(* CODESYS project twinCellBalancedProduction.export

Project tree, tasks and I/O mapping:
  Device : CODESYS Control Win V3 x64, CODESYS, version 3.5.22.30
    application Application
      libraries: Standard, 3.5.22.0 (System)
      task MainTask (cyclic, interval t#20ms, priority 1) calls PLC_PRG
      data type E_MachiningCellState
      data type E_PairCoordinatorState
      global variables Commands
      global variables FIO
      function block FB_MachiningCell [ST]
      function block FB_OperatorControl [ST]
      function block FB_PairCoordinator [ST]
      function block FB_ThroughputCounter [ST]
      program PLC_PRG [ST]
      Symbols
*)

// Device/Application/E_MachiningCellState
{attribute 'qualified_only'}
{attribute 'strict'}
TYPE E_MachiningCellState :
(
    Stopped          := 0,
    Ready            := 10,
    FeedingRaw       := 20,
    WaitingForPickup := 30,
    Processing       := 40,
    Complete         := 50,
    Faulted          := 900
);
END_TYPE

// Device/Application/E_PairCoordinatorState
{attribute 'qualified_only'}
{attribute 'strict'}
TYPE E_PairCoordinatorState :
(
    Stopped          := 0,
    Ready            := 10,
    WaitPairComplete := 20,
    MergeClearance   := 30,
    Faulted          := 900
);
END_TYPE

// Device/Application/Commands
{attribute 'qualified_only'}
VAR_GLOBAL
    // Temporary operator controls from the CODESYS watch list.
    // These can later be written by an HMI without changing the plant logic.
    xStartPB : BOOL;
    xStopPB  : BOOL;
    xResetPB : BOOL;
END_VAR

// Device/Application/FIO
{attribute 'qualified_only'}
VAR_GLOBAL
    // =========================================================
    // INPUTS FROM FACTORY I/O — Factory I/O writes, PLC reads
    // =========================================================

    // Lid machining cell
    xLidsAtEntry          : BOOL;
    xLidsAtExit           : BOOL;
    xLidsCenterBusy       : BOOL;
    xLidsCenterHasError   : BOOL;
    xLidsCenterOpened     : BOOL;
    diLidsCenterProgress  : DINT;

    // Base machining cell
    xBasesAtEntry         : BOOL;
    xBasesAtExit          : BOOL;
    xBasesCenterBusy      : BOOL;
    xBasesCenterHasError  : BOOL;
    xBasesCenterOpened    : BOOL;
    diBasesCenterProgress : DINT;
	
	// Total parts processed to removal stage
	diTotalPartsCounterDisplay : DINT;
	xTotalPartsAtRemoval       : BOOL;
	
	// Twin Cell operator-panel inputs
	xTwinCellAutoModeSelected   : BOOL;
	xTwinCellEmergencyStop      : BOOL;
	xTwinCellManualModeSelected : BOOL;
	xTwinCellResetPB            : BOOL;
	xTwinCellStartPB            : BOOL;
	xTwinCellStopPB             : BOOL;

    // Factory I/O simulation status
    xFactoryIOPaused    : BOOL;
    xFactoryIOReset     : BOOL;
    xFactoryIORunning   : BOOL;
    rFactoryIOTimeScale : REAL;


    // =========================================================
    // OUTPUTS TO FACTORY I/O — PLC writes, Factory I/O reads
    // =========================================================

    // Lid machining cell
    xLidsCenterProduceLidsCmd : BOOL;
    xLidsCenterStartCmd       : BOOL;
    xLidsCenterStopCmd        : BOOL;
    xLidsCenterResetCmd       : BOOL;
    xLidsEmitterCmd           : BOOL;
    xLidsRawConveyorCmd       : BOOL;
    xLidsExitConveyor1Cmd     : BOOL;
    xLidsExitConveyor2Cmd     : BOOL;
    diLidsCounterDisplay      : DINT;

    // Base machining cell
    xBasesCenterProduceLidsCmd : BOOL;
    xBasesCenterStartCmd       : BOOL;
    xBasesCenterStopCmd        : BOOL;
    xBasesCenterResetCmd       : BOOL;
    xBasesEmitterCmd           : BOOL;
    xBasesRawConveyorCmd       : BOOL;
    xBasesExitConveyor1Cmd     : BOOL;
    xBasesExitConveyor2Cmd     : BOOL;
    diBasesCounterDisplay      : DINT;

    // Shared outfeed
    xExitConveyorCmd : BOOL;
    xRemoverCmd      : BOOL;

    // Optional Factory I/O simulation control
    diFactoryIOCameraPositionCmd : DINT;
    xFactoryIOPauseCmd           : BOOL;
    xFactoryIOResetCmd           : BOOL;
    xFactoryIORunCmd             : BOOL;
	
	// Twin Cell operator-panel outputs
	diTwinCellBasesCounterDisplay : DINT;
	diTwinCellLidsCounterDisplay  : DINT;
	
	xTwinCellResetLightCmd        : BOOL;
	xTwinCellStartLightCmd        : BOOL;
	xTwinCellStopLightCmd         : BOOL;
END_VAR

// Device/Application/PLC_PRG
PROGRAM PLC_PRG
VAR
    // Function-block instances
    fbOperator    : FB_OperatorControl;
    fbCoordinator : FB_PairCoordinator;
    fbLidsCell    : FB_MachiningCell;
    fbBasesCell   : FB_MachiningCell;
	fbStopOutfeedClearance : TON;
	fbThroughputCounter : FB_ThroughputCounter;


    // Plant-level control
    xEnablePlant              : BOOL;
	xPlantFaulted             : BOOL;
	xRecoveryResetRequired    : BOOL;
	xResetPulse               : BOOL;
	xResetRequired            : BOOL;
	xRunLatched               : BOOL;
	xStopPending              : BOOL;


    // Coordinator handshakes
    xLidsRequest  : BOOL;
    xBasesRequest : BOOL;

    xLidsReady  : BOOL;
    xBasesReady : BOOL;

    xLidsDone  : BOOL;
    xBasesDone : BOOL;


    // Fault aggregation
    xLidsFaulted       : BOOL;
    xBasesFaulted      : BOOL;
    xCoordinatorFaulted : BOOL;

    uiLidsFaultCode  : UINT;
    uiBasesFaultCode : UINT;


    // Machining-centre commands
    xLidsProduceLidsCmd  : BOOL;
    xLidsStartCmd        : BOOL;
    xLidsStopCmd         : BOOL;
    xLidsResetCmd        : BOOL;
    xLidsRawConveyorCmd  : BOOL;

    xBasesProduceLidsCmd : BOOL;
    xBasesStartCmd       : BOOL;
    xBasesStopCmd        : BOOL;
    xBasesResetCmd       : BOOL;
    xBasesRawConveyorCmd : BOOL;


    // Production totals
    diLidsCount      : DINT;
    diBasesCount     : DINT;
    diPairsCompleted : DINT;
	diTotalPartsCount : DINT;


    // Online state diagnostics
    eLidsState :
        E_MachiningCellState;

    eBasesState :
        E_MachiningCellState;

    eCoordinatorState :
        E_PairCoordinatorState;
END_VAR

// =============================================================
// 1. PLANT FAULT STATUS FROM THE PREVIOUS PLC SCAN
// =============================================================

xPlantFaulted :=
    xBasesFaulted
    OR xCoordinatorFaulted
    OR xLidsFaulted;

// Preserve the pre-reset recovery requirement for the complete
// 500 ms reset pulse.
IF NOT xResetPulse THEN
    xRecoveryResetRequired :=
        xResetRequired;
END_IF;

// =============================================================
// 2. TWIN CELL OPERATOR CONTROL
// =============================================================
// The final counter sensor is positioned immediately before
// removal. Wait until both expected parts have passed it,
// the sensor has cleared, and the outfeed has run for another
// two seconds before completing a controlled stop.

fbStopOutfeedClearance(
    IN :=
        xStopPending
        AND (eCoordinatorState = E_PairCoordinatorState.Ready)
        AND (diTotalPartsCount >= (diPairsCompleted * DINT#2))
        AND FIO.xTotalPartsAtRemoval,
    PT :=
        T#2S
);

fbOperator(
    xAutoModeSelected :=
        FIO.xTwinCellAutoModeSelected,

    xEmergencyStop :=
        NOT FIO.xTwinCellEmergencyStop,

    xFactoryIOPaused :=
        FIO.xFactoryIOPaused,

    xFactoryIORunning :=
        FIO.xFactoryIORunning,

    xManualModeSelected :=
        FIO.xTwinCellManualModeSelected,

    xPlantFaulted :=
        xPlantFaulted,

    xResetPB :=
        Commands.xResetPB
        OR FIO.xFactoryIOReset
        OR FIO.xTwinCellResetPB,

    xSafeToStop :=
    	fbStopOutfeedClearance.Q,

    xStartPB :=
        Commands.xStartPB
        OR FIO.xTwinCellStartPB,

    xStopPB :=
        Commands.xStopPB
        OR NOT FIO.xTwinCellStopPB,

    xEnablePlant =>
        xEnablePlant,

    xResetPulse =>
        xResetPulse,

    xResetRequired =>
        xResetRequired,

    xRunLatched =>
        xRunLatched,

    xStopPending =>
        xStopPending
);

// =============================================================
// 3. PAIRED-PRODUCTION COORDINATOR
// =============================================================

fbCoordinator(
    xEnable :=
        xEnablePlant,

    xReset :=
        xResetPulse,

    xAnyFault :=
        xLidsFaulted
        OR xBasesFaulted,

    xLidsReady :=
        xLidsReady,

    xBasesReady :=
        xBasesReady,

    xLidsDone :=
        xLidsDone,

    xBasesDone :=
        xBasesDone,

    tMergeClearance :=
        T#2S,
		
	xAllowNewPair :=
    	NOT xStopPending,

    xLidsRequest =>
        xLidsRequest,

    xBasesRequest =>
        xBasesRequest,

    xFaulted =>
        xCoordinatorFaulted,

    diPairsCompleted =>
        diPairsCompleted,

    eState =>
        eCoordinatorState
);


// =============================================================
// 4. LID MACHINING CELL
// =============================================================

fbLidsCell(
    xEnable :=
        xEnablePlant,

    xReset :=
        xResetPulse,

    xRequest :=
        xLidsRequest,

    xProduceLids :=
        TRUE,

    xAtEntry := NOT FIO.xLidsAtEntry,

    xAtExit := NOT FIO.xLidsAtExit,

    xBusy :=
        FIO.xLidsCenterBusy,

    xHasError :=
        FIO.xLidsCenterHasError,

    xOpened :=
        FIO.xLidsCenterOpened,

    diProgress :=
        FIO.diLidsCenterProgress,

    tFeedTimeout :=
        T#15S,

    tPickupTimeout :=
        T#15S,

    tProcessTimeout :=
        T#90S,

    tExitClearTimeout :=
        T#10S,

    xReady =>
        xLidsReady,

    xDone =>
        xLidsDone,

    xFaulted =>
        xLidsFaulted,

    uiFaultCode =>
        uiLidsFaultCode,

    diCount =>
        diLidsCount,

    eState =>
        eLidsState,

    xRawConveyorCmd =>
        xLidsRawConveyorCmd,

    xProduceLidsCmd =>
        xLidsProduceLidsCmd,

    xStartCmd =>
        xLidsStartCmd,

    xStopCmd =>
        xLidsStopCmd,

    xResetCmd =>
        xLidsResetCmd
);


// =============================================================
// 5. BASE MACHINING CELL
// Same FB, but its product-selection input is FALSE.
// =============================================================

fbBasesCell(
    xEnable :=
        xEnablePlant,

    xReset :=
        xResetPulse,

    xRequest :=
        xBasesRequest,

    xProduceLids :=
        FALSE,

    xAtEntry := NOT FIO.xBasesAtEntry,

    xAtExit := NOT FIO.xBasesAtExit,

    xBusy :=
        FIO.xBasesCenterBusy,

    xHasError :=
        FIO.xBasesCenterHasError,

    xOpened :=
        FIO.xBasesCenterOpened,

    diProgress :=
        FIO.diBasesCenterProgress,

    tFeedTimeout :=
        T#15S,

    tPickupTimeout :=
        T#15S,

    tProcessTimeout :=
        T#90S,

    tExitClearTimeout :=
        T#10S,

    xReady =>
        xBasesReady,

    xDone =>
        xBasesDone,

    xFaulted =>
        xBasesFaulted,

    uiFaultCode =>
        uiBasesFaultCode,

    diCount =>
        diBasesCount,

    eState =>
        eBasesState,

    xRawConveyorCmd =>
        xBasesRawConveyorCmd,

    xProduceLidsCmd =>
        xBasesProduceLidsCmd,

    xStartCmd =>
        xBasesStartCmd,

    xStopCmd =>
        xBasesStopCmd,

    xResetCmd =>
        xBasesResetCmd
);

// =============================================================
// 6. FINAL THROUGHPUT COUNTER
//
// Retroreflective sensors are TRUE while the beam is clear.
// Invert the raw signal so xDetected becomes TRUE when a part
// interrupts the beam.
// =============================================================

fbThroughputCounter(
    xDetected :=
        NOT FIO.xTotalPartsAtRemoval,

    xReset :=
        xResetPulse,

    diTotalCount =>
        diTotalPartsCount
);


// Refresh the aggregate after this scan's equipment execution.
xPlantFaulted :=
    xLidsFaulted
    OR xBasesFaulted
    OR xCoordinatorFaulted;
	
// =============================================================
// 7. FACTORY I/O OUTPUT BOUNDARY
// Internal equipment commands are mapped to external OPC tags here.
// =============================================================


// -------------------------------------------------------------
// Lid machining centre
// -------------------------------------------------------------

FIO.xLidsCenterProduceLidsCmd :=
    xLidsProduceLidsCmd;

FIO.xLidsCenterStartCmd :=
    xLidsStartCmd;

FIO.xLidsCenterStopCmd :=
    xLidsStopCmd;

FIO.xLidsCenterResetCmd :=
    xLidsResetCmd;

FIO.xLidsRawConveyorCmd :=
    xLidsRawConveyorCmd;


// -------------------------------------------------------------
// Base machining centre
// -------------------------------------------------------------

FIO.xBasesCenterProduceLidsCmd :=
    xBasesProduceLidsCmd;

FIO.xBasesCenterStartCmd :=
    xBasesStartCmd;

FIO.xBasesCenterStopCmd :=
    xBasesStopCmd;

FIO.xBasesCenterResetCmd :=
    xBasesResetCmd;

FIO.xBasesRawConveyorCmd :=
    xBasesRawConveyorCmd;


// -------------------------------------------------------------
// Outfeed conveyors
//
// These run continuously while the plant is enabled. Pair
// coordination supplies the collision prevention at the merge.
// -------------------------------------------------------------

FIO.xLidsExitConveyor1Cmd :=
    xEnablePlant;

FIO.xLidsExitConveyor2Cmd :=
    xEnablePlant;

FIO.xBasesExitConveyor1Cmd :=
    xEnablePlant;

FIO.xBasesExitConveyor2Cmd :=
    xEnablePlant;

FIO.xExitConveyorCmd :=
    xEnablePlant;


// -------------------------------------------------------------
// Emitters and remover
//
// These are currently forced ON inside the supplied Factory I/O
// scene. The mappings are still complete for a later unforced V2.
// -------------------------------------------------------------

FIO.xLidsEmitterCmd :=
    xEnablePlant;

FIO.xBasesEmitterCmd :=
    xEnablePlant;

FIO.xRemoverCmd :=
    xEnablePlant;


// -------------------------------------------------------------
// Scene-mounted integer displays
// -------------------------------------------------------------

FIO.diLidsCounterDisplay :=
    diLidsCount;

FIO.diBasesCounterDisplay :=
    diBasesCount;
	
FIO.diTwinCellBasesCounterDisplay :=
    diBasesCount;

FIO.diTwinCellLidsCounterDisplay :=
    diLidsCount;
	
FIO.diTotalPartsCounterDisplay :=
    diTotalPartsCount;


// -------------------------------------------------------------
// Factory I/O simulation control
//
// Plant Reset resets PLC sequence and physical scene together.
// Run/Pause/Camera remain manually controlled for V1.
// -------------------------------------------------------------

FIO.xFactoryIOResetCmd :=
    xResetPulse
	AND xRecoveryResetRequired;

FIO.xFactoryIORunCmd :=
    FALSE;

FIO.xFactoryIOPauseCmd :=
    FALSE;

FIO.diFactoryIOCameraPositionCmd :=
    0;
	
	
FIO.xTwinCellResetLightCmd :=
    xResetRequired
    OR xPlantFaulted;

FIO.xTwinCellStartLightCmd :=
    xEnablePlant
    AND NOT xStopPending;

FIO.xTwinCellStopLightCmd :=
    NOT xRunLatched
    OR xStopPending;

END_PROGRAM

// Device/Application/FB_OperatorControl
FUNCTION_BLOCK FB_OperatorControl
VAR_INPUT
    xAutoModeSelected   : BOOL;
    xEmergencyStop      : BOOL;
    xFactoryIOPaused    : BOOL;
    xFactoryIORunning   : BOOL;
    xManualModeSelected : BOOL;
    xPlantFaulted       : BOOL;
    xResetPB            : BOOL;
    xSafeToStop         : BOOL;
    xStartPB            : BOOL;
    xStopPB             : BOOL;
END_VAR

VAR_OUTPUT
    xEnablePlant   : BOOL;
    xResetPulse    : BOOL;
    xResetRequired : BOOL := TRUE;
    xRunLatched    : BOOL;
    xStopPending   : BOOL;
END_VAR

VAR
    fbResetPulse  : TP;
    rtReset       : R_TRIG;
    rtStart       : R_TRIG;
    rtStop        : R_TRIG;
    xAutoModeValid : BOOL;
END_VAR

// =============================================================
// EDGE DETECTION
// =============================================================

rtReset(CLK := xResetPB);
rtStart(CLK := xStartPB);
rtStop(CLK := xStopPB);

// =============================================================
// OPERATING-MODE VALIDATION
//
// Exactly one selector position must be active.
// =============================================================

xAutoModeValid :=
    xAutoModeSelected
    AND NOT xManualModeSelected;

// A 500 ms pulse survives the CODESYS-Kepware-OPC-Factory I/O path.
// Reset is blocked while the emergency stop is active.
fbResetPulse(
    IN :=
        rtReset.Q
        AND NOT xEmergencyStop,
    PT := T#500MS
);

xResetPulse :=
    fbResetPulse.Q
    AND NOT xEmergencyStop;

// =============================================================
// OPERATOR COMMAND PRIORITIES
// =============================================================

IF xEmergencyStop THEN

    // Emergency stop immediately disables both machining cells.
    xResetRequired := TRUE;
    xRunLatched := FALSE;
    xStopPending := FALSE;

ELSIF rtReset.Q THEN

    // Reset clears latched faults but never starts production.
    xResetRequired := FALSE;
    xRunLatched := FALSE;
    xStopPending := FALSE;

ELSIF xPlantFaulted THEN

    // A fault in either cell stops the complete paired process.
    xResetRequired := TRUE;
    xRunLatched := FALSE;
    xStopPending := FALSE;

ELSIF NOT xAutoModeValid THEN

    xRunLatched := FALSE;
    xStopPending := FALSE;

ELSIF rtStop.Q THEN

    // Stop completes the current pair before disabling production.
    IF xSafeToStop THEN
        xRunLatched := FALSE;
        xStopPending := FALSE;
    ELSE
        xStopPending := TRUE;
    END_IF;

ELSIF xStopPending AND xSafeToStop THEN

    // The completed pair has cleared the coordinated process.
    xRunLatched := FALSE;
    xStopPending := FALSE;

ELSIF rtStart.Q
AND xFactoryIORunning
AND NOT xFactoryIOPaused
AND NOT xResetRequired
AND NOT xStopPending THEN

    xRunLatched := TRUE;
    xStopPending := FALSE;

END_IF;

// =============================================================
// FINAL AUTOMATIC-SEQUENCE PERMISSION
// =============================================================

xEnablePlant :=
    xRunLatched
    AND xAutoModeValid
    AND xFactoryIORunning
    AND NOT xEmergencyStop
    AND NOT xFactoryIOPaused
    AND NOT xPlantFaulted
    AND NOT xResetRequired;

END_FUNCTION_BLOCK

// Device/Application/FB_PairCoordinator
FUNCTION_BLOCK FB_PairCoordinator
VAR_INPUT
	xAllowNewPair : BOOL;
    xEnable   : BOOL;
    xReset    : BOOL;
    xAnyFault : BOOL;

    xLidsReady  : BOOL;
    xBasesReady : BOOL;
    xLidsDone   : BOOL;
    xBasesDone  : BOOL;

    tMergeClearance : TIME := T#2S;
END_VAR

VAR_OUTPUT
    xLidsRequest  : BOOL;
    xBasesRequest : BOOL;
    xFaulted      : BOOL;

    diPairsCompleted : DINT;

    eState : E_PairCoordinatorState :=
        E_PairCoordinatorState.Stopped;
END_VAR

VAR
    fbMergeClearance : TON;
END_VAR

// The clearance timer begins only after both cells have dropped
// their Done handshakes, cleared their exit sensors and returned Ready.
fbMergeClearance(
    IN :=
        xEnable
        AND (eState = E_PairCoordinatorState.MergeClearance)
        AND xLidsReady
        AND xBasesReady,
    PT := tMergeClearance
);


// Reset returns the complete paired sequence to a known condition.
IF xReset THEN
    xFaulted := FALSE;
    diPairsCompleted := 0;

    eState := E_PairCoordinatorState.Stopped;


// Any equipment fault latches the coordinator into Faulted.
ELSIF xAnyFault THEN
    xFaulted := TRUE;

    eState := E_PairCoordinatorState.Faulted;


// Disabling the plant freezes the active coordinator state.
ELSIF xEnable THEN

    CASE eState OF

        // -----------------------------------------------------
        // First enabled scan following Reset.
        // -----------------------------------------------------
        E_PairCoordinatorState.Stopped:

            eState := E_PairCoordinatorState.Ready;


        // -----------------------------------------------------
        // A pair begins only when both cells can accept it.
        // -----------------------------------------------------
        E_PairCoordinatorState.Ready:

			IF xAllowNewPair
			AND xBasesReady
			AND xLidsReady THEN
		
				eState :=
					E_PairCoordinatorState.WaitPairComplete;
			END_IF;


        // -----------------------------------------------------
        // Requests remain held until both cells acknowledge Done.
        // The base will normally finish first and wait here.
        // -----------------------------------------------------
        E_PairCoordinatorState.WaitPairComplete:

            IF xLidsDone AND xBasesDone THEN
                diPairsCompleted :=
                    diPairsCompleted + 1;

                eState :=
                    E_PairCoordinatorState.MergeClearance;
            END_IF;


        // -----------------------------------------------------
        // Wait for both exits and the shared merge path to clear.
        // -----------------------------------------------------
        E_PairCoordinatorState.MergeClearance:

            IF fbMergeClearance.Q THEN
                eState := E_PairCoordinatorState.Ready;
            END_IF;


        // -----------------------------------------------------
        // Latched until Reset.
        // -----------------------------------------------------
        E_PairCoordinatorState.Faulted:

            xFaulted := TRUE;


    ELSE
        xFaulted := TRUE;

        eState := E_PairCoordinatorState.Faulted;
    END_CASE;

END_IF;


// Held request/acknowledge handshake.
//
// Both requests are asserted together and disappear only when
// the coordinator leaves WaitPairComplete.
xLidsRequest :=
    xEnable
    AND NOT xFaulted
    AND
    (eState =
        E_PairCoordinatorState.WaitPairComplete);

xBasesRequest := xLidsRequest;

END_FUNCTION_BLOCK

// Device/Application/FB_MachiningCell
FUNCTION_BLOCK FB_MachiningCell
VAR_INPUT
    // Plant control
    xEnable      : BOOL;
    xReset       : BOOL;
    xRequest     : BOOL;
    xProduceLids : BOOL;

    // Factory I/O feedback
    xAtEntry   : BOOL;
    xAtExit    : BOOL;
    xBusy      : BOOL;
    xHasError  : BOOL;
    xOpened    : BOOL;
    diProgress : DINT;

    // Initial commissioning limits
    tFeedTimeout      : TIME := T#15S;
    tPickupTimeout    : TIME := T#15S;
    tProcessTimeout   : TIME := T#30S;
    tExitClearTimeout : TIME := T#10S;
END_VAR

VAR_OUTPUT
    // Handshake and diagnostics
    xReady      : BOOL;
    xDone       : BOOL;
    xFaulted    : BOOL;
    uiFaultCode : UINT;
    diCount     : DINT;

    eState : E_MachiningCellState :=
        E_MachiningCellState.Stopped;

    // Commands to Factory I/O
    xRawConveyorCmd : BOOL;
    xProduceLidsCmd : BOOL;
    xStartCmd       : BOOL;
    xStopCmd        : BOOL;
    xResetCmd       : BOOL;
END_VAR

VAR
    fbFeedTimeout      : TON;
    fbPickupTimeout    : TON;
    fbProcessTimeout   : TON;
    fbExitClearTimeout : TON;
END_VAR

// =============================================================
// STATE TIMER EXECUTION
// Timers are called every scan and enabled only in their state.
// =============================================================

fbFeedTimeout(
    IN :=
        xEnable
        AND (eState = E_MachiningCellState.FeedingRaw)
        AND NOT xAtEntry,
    PT := tFeedTimeout
);

fbPickupTimeout(
    IN :=
        xEnable
        AND (eState = E_MachiningCellState.WaitingForPickup)
        AND NOT xBusy,
    PT := tPickupTimeout
);

fbProcessTimeout(
    IN :=
        xEnable
        AND (eState = E_MachiningCellState.Processing)
        AND NOT xAtExit,
    PT := tProcessTimeout
);

fbExitClearTimeout(
    IN :=
        xEnable
        AND (eState = E_MachiningCellState.Complete)
        AND xAtExit,
    PT := tExitClearTimeout
);


// =============================================================
// DEFAULT OUTPUTS
// Every output receives a known value at the start of each scan.
// =============================================================

xReady := FALSE;
xDone := FALSE;
xRawConveyorCmd := FALSE;

xProduceLidsCmd := xProduceLids;

xStartCmd := FALSE;

xStopCmd :=
    (NOT xEnable OR xFaulted)
    AND NOT xReset;

xResetCmd := xReset;


// =============================================================
// RESET AND FAULT PRIORITIES
// =============================================================

// Reset clears the internal sequence and completed-product count.
IF xReset THEN
    xFaulted := FALSE;
    uiFaultCode := 0;
    diCount := 0;

    eState := E_MachiningCellState.Stopped;


// Factory I/O raises this for an incorrect item or station error.
ELSIF xHasError THEN
    xFaulted := TRUE;
    uiFaultCode := 1;

    eState := E_MachiningCellState.Faulted;


// A latched fault remains until Reset.
ELSIF xFaulted THEN
    eState := E_MachiningCellState.Faulted;


// Freeze the active sequence whenever the plant is disabled.
ELSIF xEnable THEN

    CASE eState OF

        // -----------------------------------------------------
        // Await the first plant enable after Reset.
        // -----------------------------------------------------
        E_MachiningCellState.Stopped:

            eState := E_MachiningCellState.Ready;


        // -----------------------------------------------------
        // Ready to accept one request from the coordinator.
        // Do not accept a new part while the exit is occupied.
        // -----------------------------------------------------
        E_MachiningCellState.Ready:

            xReady := NOT xAtExit;

            IF xRequest AND xReady THEN
                eState := E_MachiningCellState.FeedingRaw;
            END_IF;


        // -----------------------------------------------------
        // Move one staged raw item towards the entry bay.
        // -----------------------------------------------------
        E_MachiningCellState.FeedingRaw:

            xRawConveyorCmd := TRUE;

            IF xAtEntry THEN
                eState :=
                    E_MachiningCellState.WaitingForPickup;

            ELSIF fbFeedTimeout.Q THEN
                xFaulted := TRUE;
                uiFaultCode := 101; // No material at entry.

                eState := E_MachiningCellState.Faulted;
            END_IF;


        // -----------------------------------------------------
        // Wait for the robot to collect the detected material.
        //
        // Busy or the falling entry signal confirms pickup.
        // -----------------------------------------------------
       E_MachiningCellState.WaitingForPickup:

			// Continue carrying the blank beyond the external sensor
			// and into the machining centre's true pickup bay.
			xRawConveyorCmd := TRUE;
			xStartCmd := TRUE;
		
			IF xBusy THEN
				eState := E_MachiningCellState.Processing;
		
			ELSIF fbPickupTimeout.Q THEN
				xFaulted := TRUE;
				uiFaultCode := 102;
		
				eState := E_MachiningCellState.Faulted;
			END_IF;


        // -----------------------------------------------------
        // Wait until the finished product reaches the exit.
        // The state transition itself provides one-shot counting.
        // -----------------------------------------------------
        E_MachiningCellState.Processing:

            IF xAtExit THEN
                diCount := diCount + 1;

                eState := E_MachiningCellState.Complete;

            ELSIF fbProcessTimeout.Q THEN
                xFaulted := TRUE;
                uiFaultCode := 103; // Product never reached exit.

                eState := E_MachiningCellState.Faulted;
            END_IF;


        // -----------------------------------------------------
        // Hold Done until the coordinator removes Request.
        // This handshake cannot be missed between PLC scans.
        // -----------------------------------------------------
        E_MachiningCellState.Complete:

            xDone := TRUE;

            IF fbExitClearTimeout.Q THEN
                xFaulted := TRUE;
                uiFaultCode := 104; // Exit remained obstructed.

                eState := E_MachiningCellState.Faulted;

            ELSIF NOT xRequest AND NOT xAtExit THEN
                eState := E_MachiningCellState.Ready;
            END_IF;


        // -----------------------------------------------------
        // Latched safe state.
        // -----------------------------------------------------
        E_MachiningCellState.Faulted:

            xFaulted := TRUE;


    // Corrupted or unexpected enum value.
    ELSE
        xFaulted := TRUE;
        uiFaultCode := 999;

        eState := E_MachiningCellState.Faulted;
    END_CASE;

END_IF;


// =============================================================
// FINAL OUTPUT INTERLOCK
// No state can bypass this safety layer.
// =============================================================

IF NOT xEnable OR xFaulted THEN
    xRawConveyorCmd := FALSE;
    xStartCmd := FALSE;
    xStopCmd := NOT xReset;
END_IF;


// Reset must not compete with Start or Stop.
IF xReset THEN
    xStartCmd := FALSE;
    xStopCmd := FALSE;
    xResetCmd := TRUE;
END_IF;

END_FUNCTION_BLOCK

// Device/Application/FB_ThroughputCounter
FUNCTION_BLOCK FB_ThroughputCounter

VAR_INPUT
    xDetected : BOOL;
    xReset    : BOOL;
END_VAR

VAR_OUTPUT
    diTotalCount : DINT;
END_VAR

VAR
    fbDetectedEdge : R_TRIG;
END_VAR

// Count only the rising edge of a detection.
// A part remaining over the sensor therefore counts once.
fbDetectedEdge(CLK := xDetected);

IF xReset THEN
    diTotalCount := 0;

ELSIF fbDetectedEdge.Q THEN
    diTotalCount := diTotalCount + 1;
END_IF;

END_FUNCTION_BLOCK
